// TIA Portal V17 export
// export: Created 2024-08-09T12:53:21.0635145Z, ExportSetting WithDefaults, DisplayName Totally Integrated Automation Portal, DisplayVersion V17 Update 7, DisplayName TIA Portal Openness, DisplayVersion V17 Update 7, DisplayName TIA Portal Version Control Interface, DisplayVersion V17, DisplayName STEP 7 Professional, DisplayVersion V17 Update 7, DisplayName STEP 7 Safety, DisplayVersion V17 Update 6, DisplayName WinCC Professional, DisplayVersion V17 Update 7
TYPE "S_GEST_TOUR"
// stored: IsFailsafeCompliant false
   STRUCT
      _PtSuivCharg { ExternalAccessible := 'False'; ExternalVisible := 'False'; ExternalWritable := 'False'} : "S_SuiviCommunCharg";   // Zone de suivie chargement
      _Ptzs { ExternalAccessible := 'False'; ExternalVisible := 'False'; ExternalWritable := 'False'} : "S_SuiviCommande";   // zone de suivi de lot
      _PtzsPrec { ExternalAccessible := 'False'; ExternalVisible := 'False'; ExternalWritable := 'False'} : "S_SuiviCommande";   // zone de suivi de lot
      _PtzsPrec1 { ExternalAccessible := 'False'; ExternalVisible := 'False'; ExternalWritable := 'False'} : "S_SuiviCommande";   // zone de suivi de lot
      _ChargCommun : "S_ChargCommun";
      Dial_Def { ExternalAccessible := 'False'; ExternalVisible := 'False'; ExternalWritable := 'False'} : "S_DIALOG_DEF";
      _ListeTaFinChargCommande { ExternalAccessible := 'False'; ExternalVisible := 'False'; ExternalWritable := 'False'} : Array[0.."T_MAX_AMONTAVAL"] of "S_TacheNiv";   // Liste des niveaux tester pour attendre la fin de chargement de la commande
      _DebutLecPlan { ExternalAccessible := 'False'; ExternalVisible := 'False'; ExternalWritable := 'False'} : Date_And_Time;
      _TpsPicke { ExternalAccessible := 'False'; ExternalVisible := 'False'; ExternalWritable := 'False'} : Date_And_Time;
      _TpLecPlanAuto { ExternalAccessible := 'False'; ExternalVisible := 'False'; ExternalWritable := 'False'} : Time;   // Tempo entre 2 lecture planning automatique
      NumAutrePont { ExternalAccessible := 'False'; ExternalVisible := 'False'; ExternalWritable := 'False'} : Array[0.."MAX_PONT"] of SInt;
      _Badge { ExternalAccessible := 'False'; ExternalVisible := 'False'; ExternalWritable := 'False'} : String;   // Badge demande
      _SauveBadge { ExternalAccessible := 'False'; ExternalVisible := 'False'; ExternalWritable := 'False'} : String;
      _Camion { ExternalAccessible := 'False'; ExternalVisible := 'False'; ExternalWritable := 'False'} : String;   // camion demande
      _Chauffeur { ExternalAccessible := 'False'; ExternalVisible := 'False'; ExternalWritable := 'False'} : String;   // chauffeur demande
      _NoTour { ExternalAccessible := 'False'; ExternalVisible := 'False'; ExternalWritable := 'False'} : String;   // Numeo de tournee demande
      _TolSup { ExternalAccessible := 'False'; ExternalVisible := 'False'; ExternalWritable := 'False'} : Real;   // tolerence superieur de chargement par defaut
      _TolInf { ExternalAccessible := 'False'; ExternalVisible := 'False'; ExternalWritable := 'False'} : Real;   // tolerence inferieur de chargement par defaut
      _PoidsMaxCamions { ExternalAccessible := 'False'; ExternalVisible := 'False'; ExternalWritable := 'False'} : Real;   // Poids maximum d'un Camion
      _TaCharg1 { ExternalAccessible := 'False'; ExternalVisible := 'False'; ExternalWritable := 'False'} : SInt;   // No de tache boucle chargement 1
      _TaChargCompo { ExternalAccessible := 'False'; ExternalVisible := 'False'; ExternalWritable := 'False'} : SInt;   // No de tache boucle chargement composant
      _TaDosCompo { ExternalAccessible := 'False'; ExternalVisible := 'False'; ExternalWritable := 'False'} : SInt;   // No de tache boucle dosage composant
      _TaPositCam { ExternalAccessible := 'False'; ExternalVisible := 'False'; ExternalWritable := 'False'} : SInt;   // No de tache boucle positionnement Camion
      _DemTour { ExternalAccessible := 'False'; ExternalVisible := 'False'; ExternalWritable := 'False'} : USInt;
      _ZoneSuiv { ExternalAccessible := 'False'; ExternalVisible := 'False'; ExternalWritable := 'False'} : SInt;
      _ValidLecPlan : Bool;   // Validation Lecture planning
      _ValidBadge : Bool;   // Validation gestion badge
      _ChargBenne { ExternalAccessible := 'False'; ExternalVisible := 'False'; ExternalWritable := 'False'} : Bool;   // chargement avec benne
      _PreDosCompo { ExternalAccessible := 'False'; ExternalVisible := 'False'; ExternalWritable := 'False'} : Bool;   // Predosage des composants
      _DemLectCharg : Bool;   // Demande lecture planning chargement
      _ValideClotureTournee { ExternalAccessible := 'False'; ExternalVisible := 'False'; ExternalWritable := 'False'} : Bool;   // validation cloture tourne par automatisme -1 cloture avec dialogue_def -2 sans dialogue_def
      _AffMessAutrePont { ExternalAccessible := 'False'; ExternalVisible := 'False'; ExternalWritable := 'False'} : Bool;   // Validation affichage message chargement sur autre pont
      _ValidLecPlanAuto { ExternalAccessible := 'False'; ExternalVisible := 'False'; ExternalWritable := 'False'} : Bool;   // Validation lecture planning automatique
      _ValidTourAuto { ExternalAccessible := 'False'; ExternalVisible := 'False'; ExternalWritable := 'False'} : Bool;   // Return de la fonction rechtour recherche dans le planning
   END_STRUCT;
   // NumAutrePont[0..9] := -1;
END_TYPE
